{attribute addProperty BoxType "EK1100-0000-0018"}
{attribute addProperty Id "Beckhoff_EQ2xxxEK1122Beckhoff_EQ2xxxEK1122_609ED8271871233.875"}
{attribute addProperty CRC "2879429967"}
{attribute addProperty SizeInBites "1871"}
{attribute addProperty SizeInBytes "233.875"}
TYPE Beckhoff_EQ2xxx_ABA09D4F EXTENDS EK1100_179A0949 :
STRUCT
	{attribute addProperty Name "Beckhoff_EQ2xxxEK1122"}
	Beckhoff_EQ2xxxEK1122 : Beckhoff_EQ2xxxEK1122_609ED827;
END_STRUCT
END_TYPE

(* stored: Version 1.2.0.0, ProductVersion 3.1.4024.9
   DUT Beckhoff_EQ2xxx_ABA09D4F: Id {46781117-705a-4015-a2e3-337f84c070a7} *)
